// TIA Portal V18 export
FUNCTION_BLOCK "_screen_SetHome"   // FB77, FBD
{ S7_Optimized_Access := 'TRUE' }
VERSION : 0.1
// stored: AutoNumber true, IsIECCheckEnabled false, IsRetainMemResEnabled false, MemoryReserve 100, SetENOAutomatically false, UDAEnableTagReadback false
   VAR
      t_z : "hmi_home_1";
      t_o1 : "hmi_home_1";
      t_o2 : "hmi_home_1";
      t_x : "hmi_home_1";
      t_y : "hmi_home_1";
      z : "hmi_home_1";
      o1 : "hmi_home_1";
      o2 : "hmi_home_1";
      x : "hmi_home_1";
      y : "hmi_home_1";
   END_VAR
BEGIN

REGION Network 1
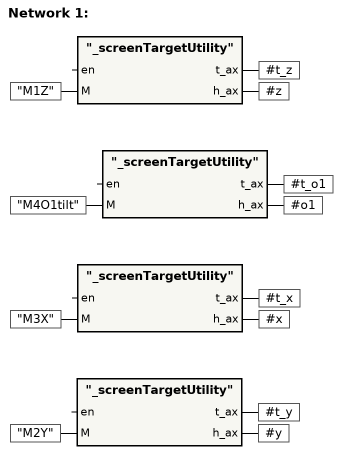
   "_screenTargetUtility"("M" := "M1Z", t_ax => #t_z, h_ax => #z);
   "_screenTargetUtility"("M" := "M4O1tilt", t_ax => #t_o1, h_ax => #o1);
   "_screenTargetUtility"("M" := "M3X", t_ax => #t_x, h_ax => #x);
   "_screenTargetUtility"("M" := "M2Y", t_ax => #t_y, h_ax => #y);
END_REGION

REGION Network 2 (SCL)
   #o2.eF := NOT "M5O2rot".xPredifCal;
   #o2.pos := "M5O2rot".POS;
   #t_o2.pos := "M5O2rot".AMANGRDB.aut_target;
END_REGION
END_FUNCTION_BLOCK
